Omron CX-Programmer project NewProject (CX-Programmer 9.61)

# PLC NewPLC1: CP1E N30

## Global symbols (name address type ; comment)
0.00 BOOL  ; ON
0.01 BOOL  ; OFF
100.00 BOOL  ; LAMP
100.01 BOOL  ; LAMP2
2 CHANNEL  ; RUN

## Program NewProgram1 (cyclic task 0)

### Section Section1

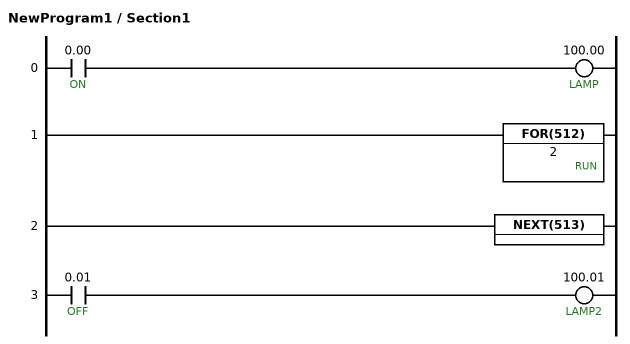
; rung 0
LD 0.00  ; ON
OUT 100.00  ; LAMP
; rung 1
FOR(512) 2  ; RUN
; rung 2
NEXT(513)
; rung 3
LD 0.01  ; OFF
OUT 100.01  ; LAMP2

### Section END
; rung 0
END(001)